Universal Robots PolyScope program: Alinear en plano vertical.urp

Program Alinear en plano vertical (installation=default directory=/home/ur/ursim-current/programs createdIn=3.15.1.106171 lastSavedIn=5.11.9.1010452 robotSerialNumber=20195599999)
Calibrated DH parameters: a=[0, -0.425, -0.3922, 0, 0, 0]; d=[0.1625, 0, 0, 0.1333, 0.0997, 0.0996]; alpha=[1.570796, 0, 0, 1.570796, -1.570796, 0]; deltaTheta=[0, 0, 0, 0, 0, 0]
BeforeStart
  Script file /home/ur/ursim-current/programs/alinearrobot.script
    | def alinearRobot(pose_actual):
    | target_pose=p[0,0,0,0,0,0]
    | rotRPY = [0,0,0]
    | rotRotvec = [0,0,0]
    | rotRPY=rotvec2rpy([pose_actual[3],pose_actual[4],pose_actual[5]])
    | rotRPY[0]=d2r(270)
    | rotRPY[1]=d2r(270)
    | rotRotvec=rpy2rotvec(rotRPY)
    | target_pose[0]=pose_actual[0]
    | target_pose[1]=pose_actual[1]
    | target_pose[2]=pose_actual[2]
    | target_pose[3]=rotRotvec[0]
    | target_pose[4]=rotRotvec[1]
    | target_pose[5]=rotRotvec[2]
    | 
    | return target_pose
    | end
  MoveJ speed 60 deg/s, acceleration 80 deg/s^2 (useActiveTCP=true) feature=Base
    Waypoint Punto_de_paso_1: TCP in base x=-173.267 y=289.864 z=340.695 mm, rx=-3.0166 ry=-0.2016 rz=0.1541 rad; joints [-84.183, -114.728, 132.722, -114.77, -84.414, -1.499] deg
    SuppressedNode
      rotacionRPY := [0,0,0]
    SuppressedNode
      rotacionRotvec := [0,0,0]
Robot Program (runOnlyOnce=true)
  Script: target=alinearRobot(get_actual_tcp_pose())
  MoveJ speed 60 deg/s, acceleration 80 deg/s^2 (useActiveTCP=true) feature=Base
    Waypoint Waypoint (Variable): variable=target
  Wait Sleep waitTime=2
  SuppressedNode
    MoveJ speed 60 deg/s, acceleration 80 deg/s^2 (useActiveTCP=true) feature=Base
      Waypoint Punto_de_paso_1: TCP in base x=-173.267 y=289.864 z=340.695 mm, rx=-3.0166 ry=-0.2016 rz=0.1541 rad; joints [-84.183, -114.728, 132.722, -114.77, -84.414, -1.499] deg
